FUNCTION_BLOCK T_CommandQueue_AddHighPriority_ReturnTrue EXTENDS T_UnitTestBase
VAR
  command : T_CommandTask;
  commandQueue : T_CommandQueue;
  myTestState, prevState : (ARRANGE, ACT, ASSERT);
  actual : BOOL := TRUE;
  expected : BOOL := TRUE;
END_VAR

CASE myTestState OF
  ARRANGE:
    myTestState := ACT;

  ACT:
    actual := commandQueue.AddHighPriority(command);
    myTestState := ASSERT;

  ASSERT:
    assertion.AssertEquals_BOOL(expected, actual, 'commandQueue.AddHighPriority = TRUE');
    myTestState := ARRANGE;
    TestFinished();
END_CASE

END_FUNCTION_BLOCK

(* stored: Version 1.1.0.1, ProductVersion 3.1.4024.12
   POU T_CommandQueue_AddHighPriority_ReturnTrue: Id {5c3b88e2-cb14-4d78-acf5-9e300df4692f}, SpecialFunc None *)
